TYPE ST_enclosure_set :
STRUCT
	by_LedBrightness 	: BYTE := 100;
END_STRUCT
END_TYPE

(* stored: Version 1.1.0.1, ProductVersion 3.1.4026.18
   DUT ST_enclosure_set: Id {06763b1f-2c5a-4d26-b542-0b98deaf1893} *)
